{attribute 'qualified_only'}
{attribute 'strict'}
TYPE E_State :
(
 	STATE_INIT,
	STATE_CONNECTING,
	STATE_RECEIVING_DATA,
	STATE_SENDING_DATA,
	STATE_PROCESSING_DATA
);
END_TYPE

(* stored: Version 1.1.0.1, ProductVersion 3.1.4024.3
   DUT E_State: Id {63a6f567-c3f9-4d8d-80e7-6dd36180d8e9} *)
